FUNCTION_BLOCK FB_SimulatedOutOpen_DG IMPLEMENTS ITF_Regelschuif_OutOpen_DG
VAR
	internalState : BOOL := FALSE;
END_VAR

METHOD set : BOOL
VAR_INPUT
	state : BOOL;
END_VAR
internalState := state;
END_METHOD

END_FUNCTION_BLOCK

(* stored: Version 1.1.0.1, ProductVersion 3.1.4026.8
   POU FB_SimulatedOutOpen_DG: Id {912669fe-b594-46ab-9d35-fdb4a26b8827}, SpecialFunc None
   Method set: Id {4e3c24d6-45b0-4602-8092-80b72458db64} *)
